TYPE ST_PU_Parameter :
STRUCT
	Regelung_PI_Kp				: REAL;
	Regelung_PI_Tn				: DINT;
	Regelung_PI_Tctr			: DINT;

	Zeit_Vorl					: DINT;
	Zeit_Nachl					: DINT;

	Stellwert_Leistung_Max		: SINT;
	Stellwert_Leistung_Min		: SINT;

	AutoQuittierung				: BOOL;
END_STRUCT
END_TYPE

(* stored: Version 1.1.0.1, ProductVersion 3.1.4024.9
   DUT ST_PU_Parameter: Id {77f9e027-acef-46af-a8aa-50e3829ebeca} *)
